FUNCTION_BLOCK FB_LineAxis
VAR_INPUT
	Execute:				ST_TriggerMode;
	System:					REFERENCE TO ST_System;
END_VAR
VAR_OUTPUT
	Moving:					BOOL;
END_VAR
VAR
END_VAR

Moving:=FALSE;

IF System.stInput.bReset  THEN
	Moving:=FALSE;
	Execute.bAuto:=Execute.bManual:=FALSE;
END_IF

IF System.stMode.stDeviceRest.bAuto THEN
	Execute.bAuto:=FALSE;
END_IF
IF System.stMode.stDeviceRest.bManual THEN
	Execute.bManual:=FALSE;
END_IF

IF System.stMode.bAutoRunning THEN
	Moving:=Execute.bAuto;
END_IF
IF System.stMode.bManual THEN
	Moving:=Execute.bManual;
END_IF

METHOD M_Jog : BOOL
VAR_INPUT
	In:				INT;//0 停止 1正转
END_VAR
CASE In OF
	0:
		Execute.bAuto:=FALSE;
	1:
		Execute.bAuto:=TRUE;
END_CASE
M_Jog:=true;
END_METHOD

END_FUNCTION_BLOCK

(* stored: Version 1.1.0.1, ProductVersion 3.1.4024.3
   POU FB_LineAxis: Id {b1eab20f-524e-4969-82ec-b988eb20465a}, SpecialFunc None
   Method M_Jog: Id {6e33dc88-29fd-4fd1-9c1a-76be6353004c} *)
